// Mitsubishi GX Works2 project: PLC_2   PLC: Q04UDV

PROGRAM MAIN
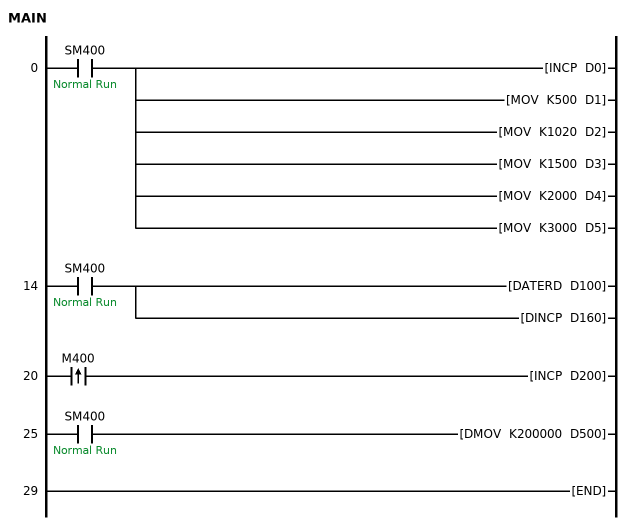
0     LD      SM400  ; Normal Run
      INCP    D0
      MOV     K500 D1
      MOV     K1020 D2
      MOV     K1500 D3
      MOV     K2000 D4
      MOV     K3000 D5
14    LD      SM400  ; Normal Run
      DATERD  D100
      DINCP   D160
20    LDP     M400
      INCP    D200
25    LD      SM400  ; Normal Run
      DMOV    K200000 D500
29    END
END_PROGRAM

PROGRAM LOSSCODE
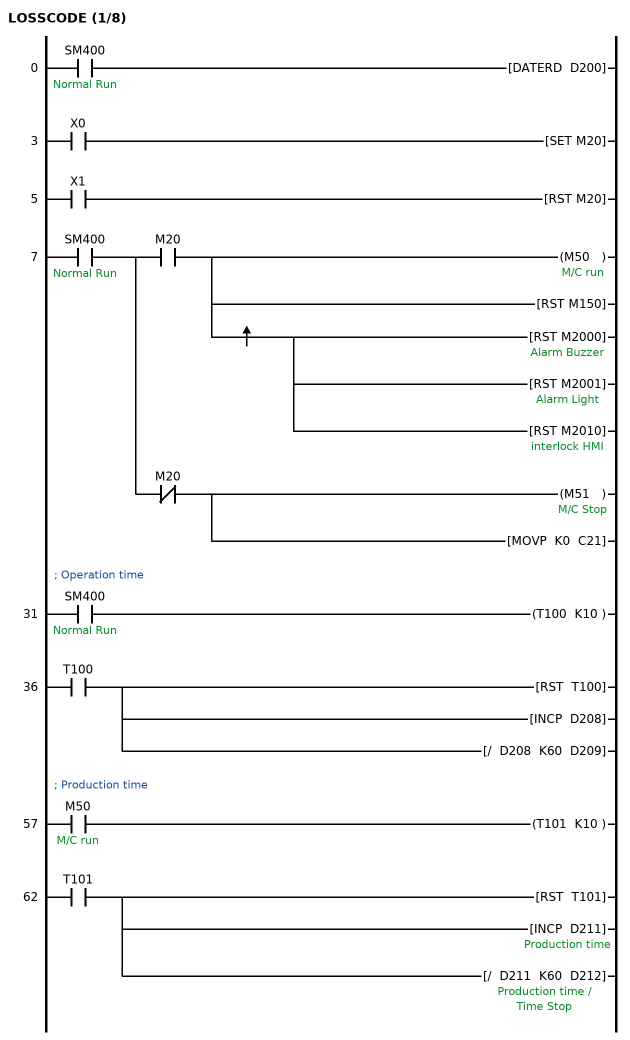
0     LD      SM400  ; Normal Run
      DATERD  D200
3     LD      X0
      SET     M20
5     LD      X1
      RST     M20
7     LD      SM400  ; Normal Run
      MPS
      AND     M20
      OUT     M50  ; M/C run
      RST     M150
      MEP
      RST     M2000  ; Alarm Buzzer
      RST     M2001  ; Alarm Light
      RST     M2010  ; interlock HMI
      MPP
      ANI     M20
      OUT     M51  ; M/C Stop
      MOVP    K0 C21
; Operation time
31    LD      SM400  ; Normal Run
      OUT     T100 K10
36    LD      T100
      RST     T100
      INCP    D208
      /       D208 K60 D209
; Production time
57    LD      M50  ; M/C run
      OUT     T101 K10
62    LD      T101
      RST     T101
      INCP    D211  ; Production time
      /       D211 K60 D212  ; Time Stop
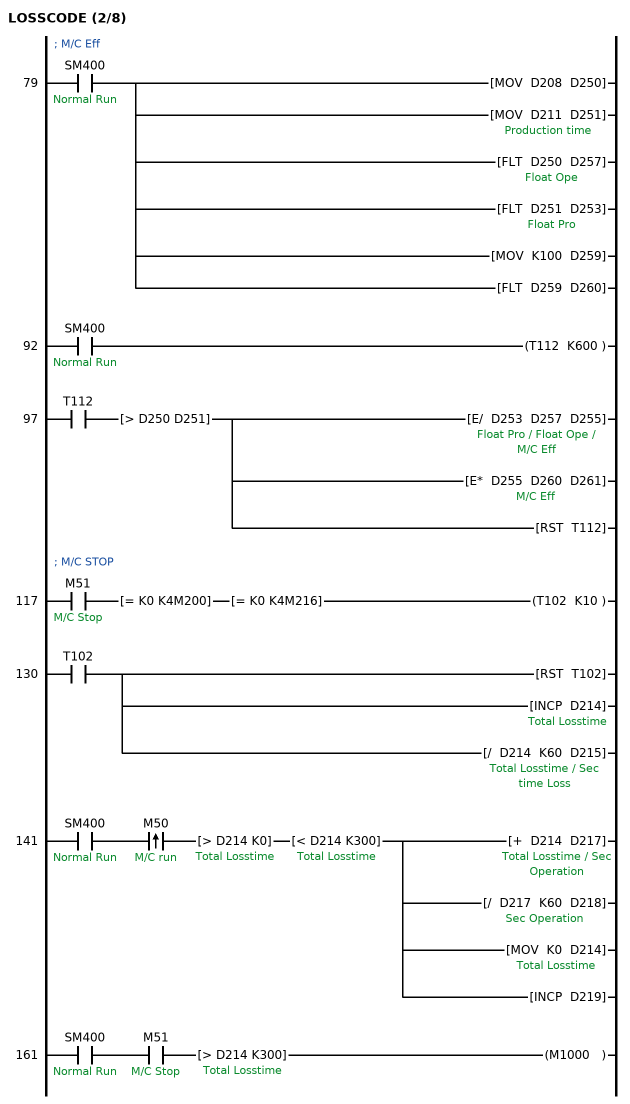
; M/C Eff
79    LD      SM400  ; Normal Run
      MOV     D208 D250
      MOV     D211 D251
      FLT     D250 D257  ; Float Ope
      FLT     D251 D253  ; Float Pro
      MOV     K100 D259
      FLT     D259 D260
92    LD      SM400  ; Normal Run
      OUT     T112 K600
97    LD      T112
      AND>    D250 D251
      E/      D253 D257 D255  ; M/C Eff
      E*      D255 D260 D261
      RST     T112
; M/C STOP
117   LD      M51  ; M/C Stop
      AND=    K0 K4M200
      AND=    K0 K4M216
      OUT     T102 K10
130   LD      T102
      RST     T102
      INCP    D214  ; Total Losstime
      /       D214 K60 D215  ; Sec time Loss
141   LD      SM400  ; Normal Run
      ANDP    M50  ; M/C run
      AND>    D214 K0  ; Total Losstime
      AND<    D214 K300  ; Total Losstime
      +       D214 D217  ; Sec Operation
      /       D217 K60 D218
      MOV     K0 D214
      INCP    D219
161   LD      SM400  ; Normal Run
      AND     M51  ; M/C Stop
      AND>    D214 K300  ; Total Losstime
      OUT     M1000
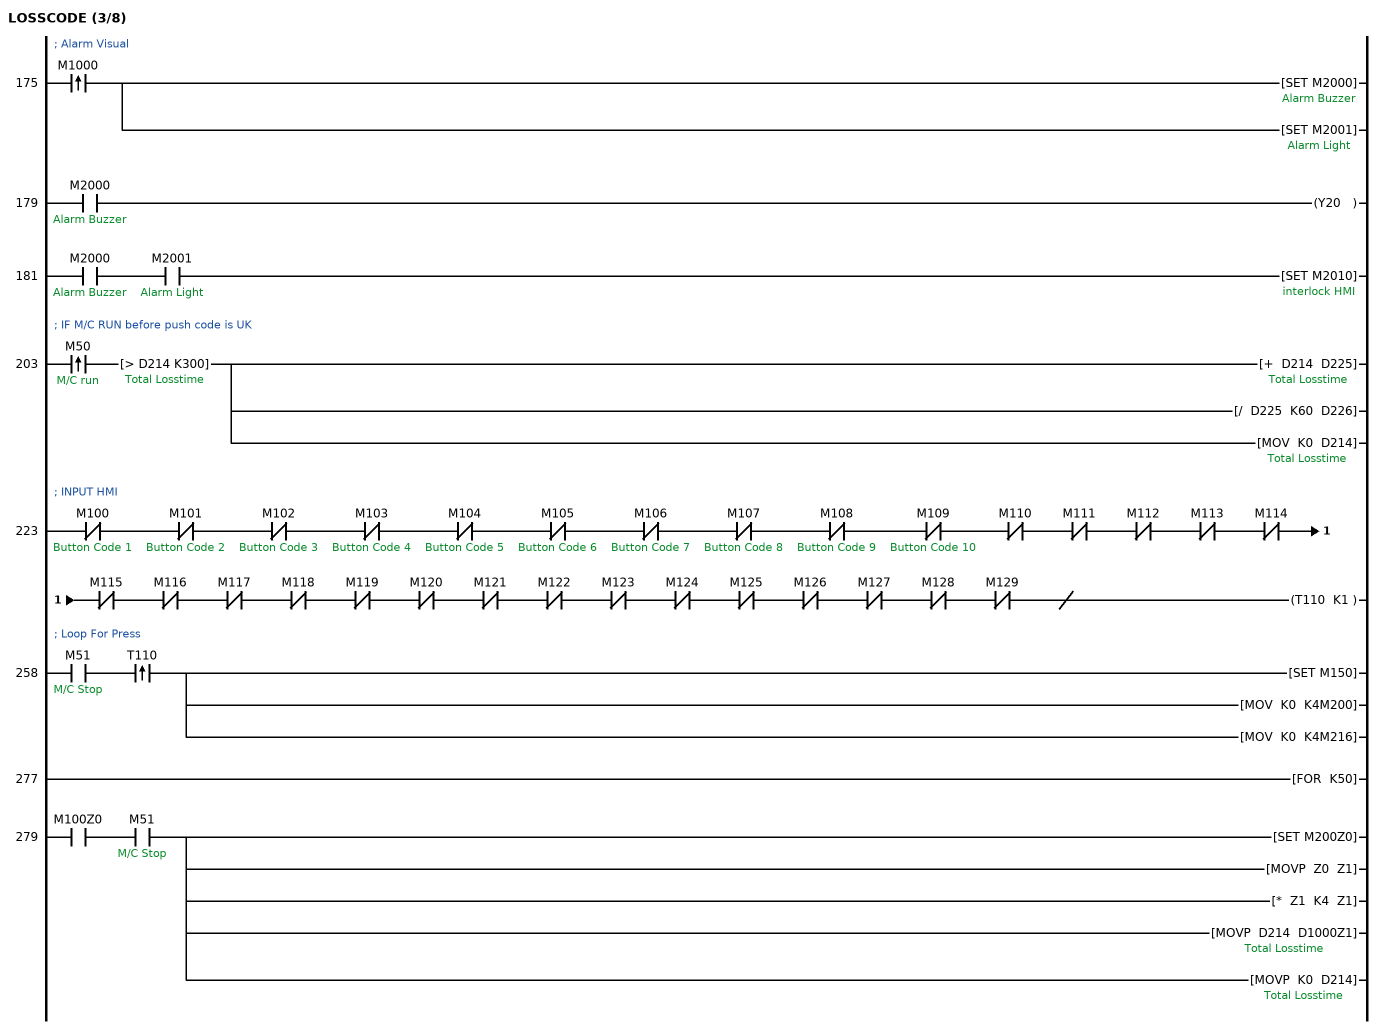
; Alarm Visual
175   LDP     M1000
      SET     M2000  ; Alarm Buzzer
      SET     M2001  ; Alarm Light
179   LD      M2000  ; Alarm Buzzer
      OUT     Y20
181   LD      M2000  ; Alarm Buzzer
      AND     M2001  ; Alarm Light
      SET     M2010  ; interlock HMI
; IF M/C RUN before push code is UK
203   LDP     M50  ; M/C run
      AND>    D214 K300  ; Total Losstime
      +       D214 D225
      /       D225 K60 D226
      MOV     K0 D214
; INPUT HMI
223   LDI     M100  ; Button Code 1
      ANI     M101  ; Button Code 2
      ANI     M102  ; Button Code 3
      ANI     M103  ; Button Code 4
      ANI     M104  ; Button Code 5
      ANI     M105  ; Button Code 6
      ANI     M106  ; Button Code 7
      ANI     M107  ; Button Code 8
      ANI     M108  ; Button Code 9
      ANI     M109  ; Button Code 10
      ANI     M110
      ANI     M111
      ANI     M112
      ANI     M113
      ANI     M114
      ANI     M115
      ANI     M116
      ANI     M117
      ANI     M118
      ANI     M119
      ANI     M120
      ANI     M121
      ANI     M122
      ANI     M123
      ANI     M124
      ANI     M125
      ANI     M126
      ANI     M127
      ANI     M128
      ANI     M129
      INV
      OUT     T110 K1
258   LD      M51  ; M/C Stop
      ANDP    T110
      SET     M150
      MOV     K0 K4M200
      MOV     K0 K4M216
; Loop For Press
277   FOR     K50
279   LD      M100Z0
      AND     M51  ; M/C Stop
      SET     M200Z0
      MOVP    Z0 Z1
      *       Z1 K4 Z1
      MOVP    D214 D1000Z1
      MOVP    K0 D214
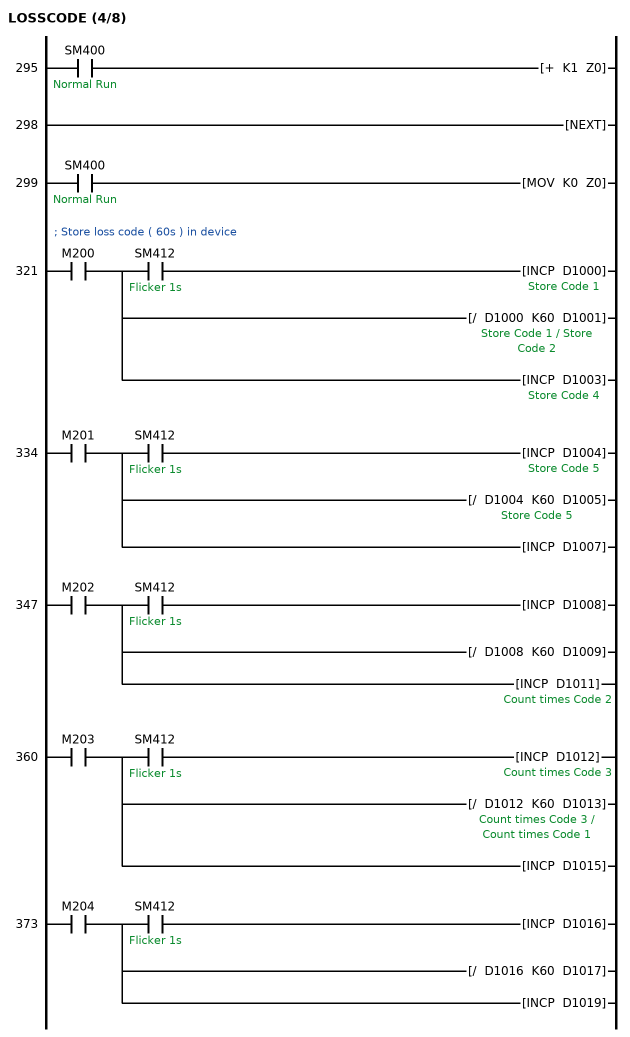
295   LD      SM400  ; Normal Run
      +       K1 Z0
298   NEXT
299   LD      SM400  ; Normal Run
      MOV     K0 Z0
; Store loss code ( 60s ) in device
321   LD      M200
      MPS
      AND     SM412  ; Flicker 1s
      INCP    D1000  ; Store Code 1
      MPP
      /       D1000 K60 D1001  ; Store Code 2
      INCP    D1003  ; Store Code 4
334   LD      M201
      MPS
      AND     SM412  ; Flicker 1s
      INCP    D1004  ; Store Code 5
      MPP
      /       D1004 K60 D1005
      INCP    D1007
347   LD      M202
      MPS
      AND     SM412  ; Flicker 1s
      INCP    D1008
      MPP
      /       D1008 K60 D1009
      INCP    D1011  ; Count times Code 2
360   LD      M203
      MPS
      AND     SM412  ; Flicker 1s
      INCP    D1012  ; Count times Code 3
      MPP
      /       D1012 K60 D1013  ; Count times Code 1
      INCP    D1015
373   LD      M204
      MPS
      AND     SM412  ; Flicker 1s
      INCP    D1016
      MPP
      /       D1016 K60 D1017
      INCP    D1019
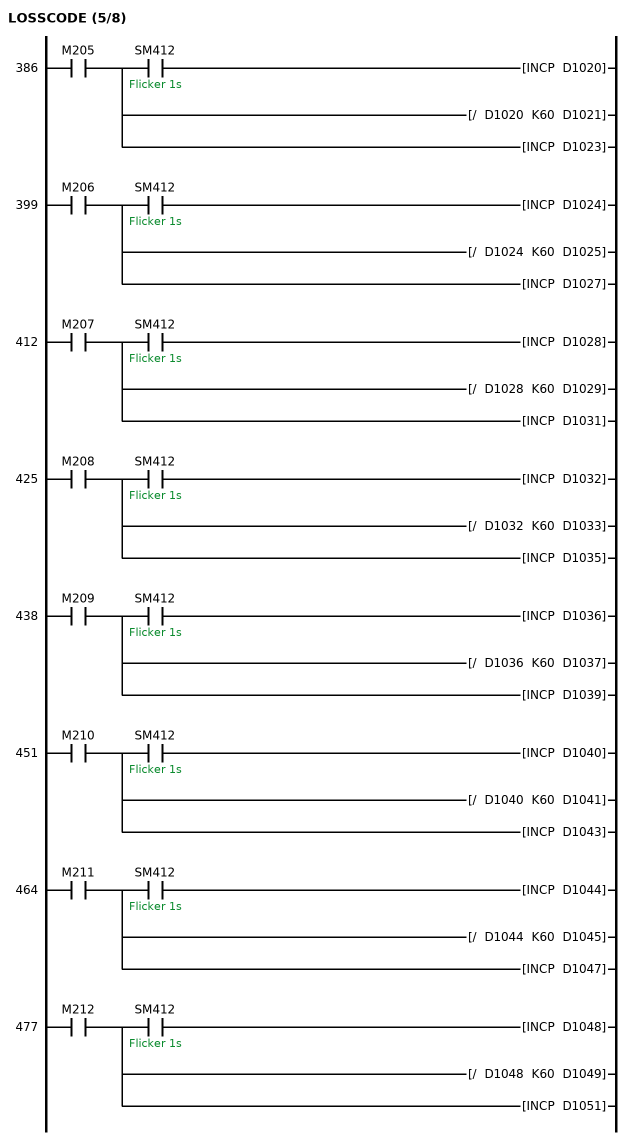
386   LD      M205
      MPS
      AND     SM412  ; Flicker 1s
      INCP    D1020
      MPP
      /       D1020 K60 D1021
      INCP    D1023
399   LD      M206
      MPS
      AND     SM412  ; Flicker 1s
      INCP    D1024
      MPP
      /       D1024 K60 D1025
      INCP    D1027
412   LD      M207
      MPS
      AND     SM412  ; Flicker 1s
      INCP    D1028
      MPP
      /       D1028 K60 D1029
      INCP    D1031
425   LD      M208
      MPS
      AND     SM412  ; Flicker 1s
      INCP    D1032
      MPP
      /       D1032 K60 D1033
      INCP    D1035
438   LD      M209
      MPS
      AND     SM412  ; Flicker 1s
      INCP    D1036
      MPP
      /       D1036 K60 D1037
      INCP    D1039
451   LD      M210
      MPS
      AND     SM412  ; Flicker 1s
      INCP    D1040
      MPP
      /       D1040 K60 D1041
      INCP    D1043
464   LD      M211
      MPS
      AND     SM412  ; Flicker 1s
      INCP    D1044
      MPP
      /       D1044 K60 D1045
      INCP    D1047
477   LD      M212
      MPS
      AND     SM412  ; Flicker 1s
      INCP    D1048
      MPP
      /       D1048 K60 D1049
      INCP    D1051
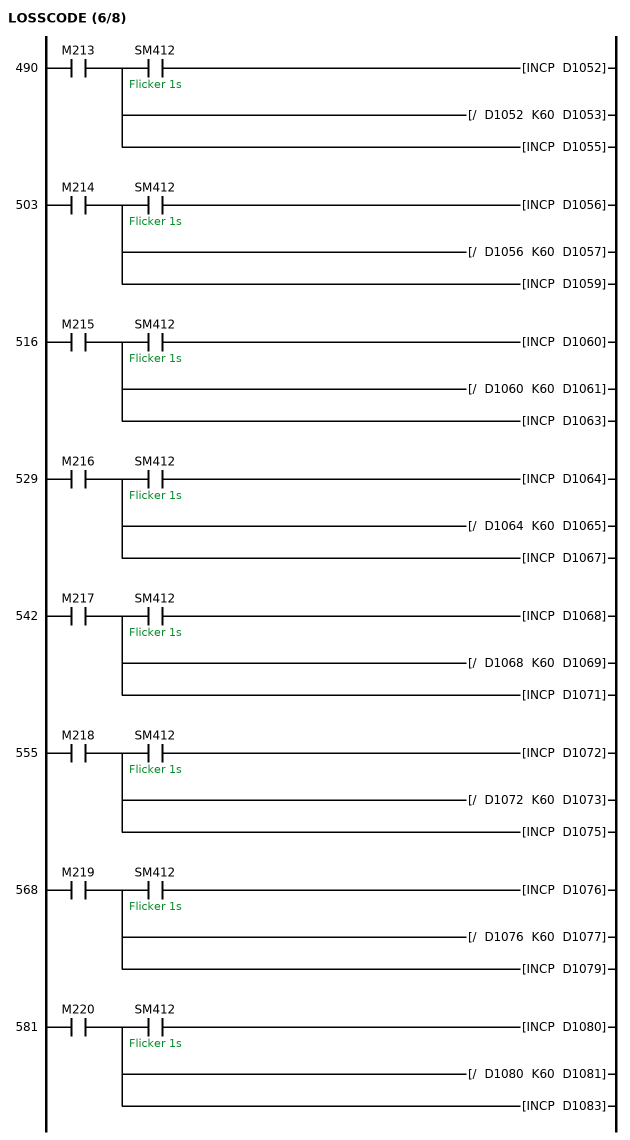
490   LD      M213
      MPS
      AND     SM412  ; Flicker 1s
      INCP    D1052
      MPP
      /       D1052 K60 D1053
      INCP    D1055
503   LD      M214
      MPS
      AND     SM412  ; Flicker 1s
      INCP    D1056
      MPP
      /       D1056 K60 D1057
      INCP    D1059
516   LD      M215
      MPS
      AND     SM412  ; Flicker 1s
      INCP    D1060
      MPP
      /       D1060 K60 D1061
      INCP    D1063
529   LD      M216
      MPS
      AND     SM412  ; Flicker 1s
      INCP    D1064
      MPP
      /       D1064 K60 D1065
      INCP    D1067
542   LD      M217
      MPS
      AND     SM412  ; Flicker 1s
      INCP    D1068
      MPP
      /       D1068 K60 D1069
      INCP    D1071
555   LD      M218
      MPS
      AND     SM412  ; Flicker 1s
      INCP    D1072
      MPP
      /       D1072 K60 D1073
      INCP    D1075
568   LD      M219
      MPS
      AND     SM412  ; Flicker 1s
      INCP    D1076
      MPP
      /       D1076 K60 D1077
      INCP    D1079
581   LD      M220
      MPS
      AND     SM412  ; Flicker 1s
      INCP    D1080
      MPP
      /       D1080 K60 D1081
      INCP    D1083
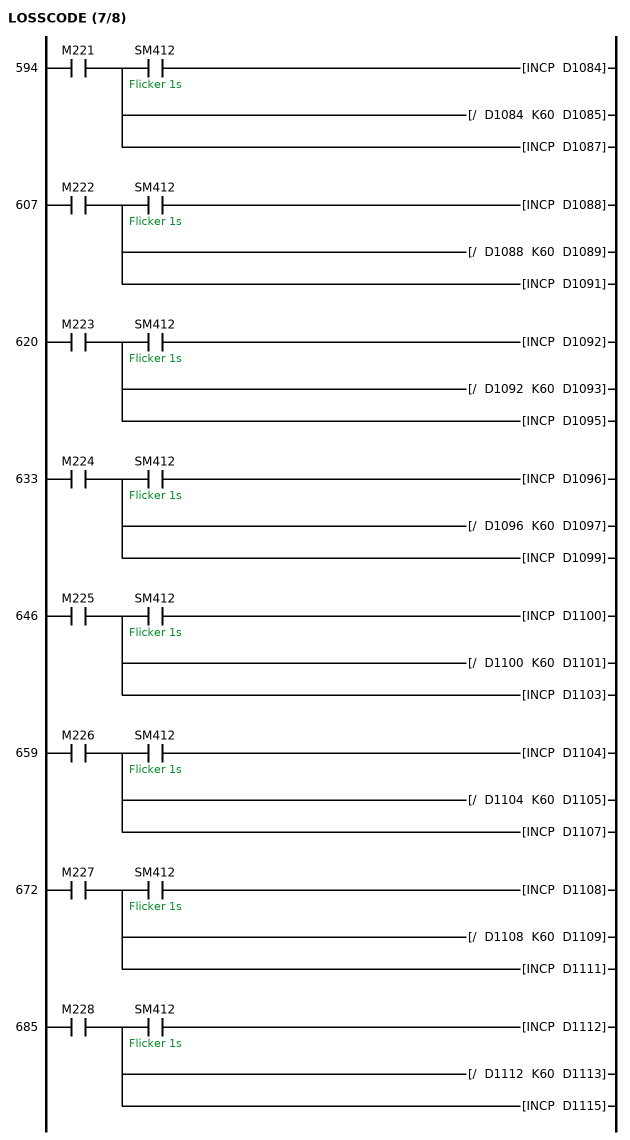
594   LD      M221
      MPS
      AND     SM412  ; Flicker 1s
      INCP    D1084
      MPP
      /       D1084 K60 D1085
      INCP    D1087
607   LD      M222
      MPS
      AND     SM412  ; Flicker 1s
      INCP    D1088
      MPP
      /       D1088 K60 D1089
      INCP    D1091
620   LD      M223
      MPS
      AND     SM412  ; Flicker 1s
      INCP    D1092
      MPP
      /       D1092 K60 D1093
      INCP    D1095
633   LD      M224
      MPS
      AND     SM412  ; Flicker 1s
      INCP    D1096
      MPP
      /       D1096 K60 D1097
      INCP    D1099
646   LD      M225
      MPS
      AND     SM412  ; Flicker 1s
      INCP    D1100
      MPP
      /       D1100 K60 D1101
      INCP    D1103
659   LD      M226
      MPS
      AND     SM412  ; Flicker 1s
      INCP    D1104
      MPP
      /       D1104 K60 D1105
      INCP    D1107
672   LD      M227
      MPS
      AND     SM412  ; Flicker 1s
      INCP    D1108
      MPP
      /       D1108 K60 D1109
      INCP    D1111
685   LD      M228
      MPS
      AND     SM412  ; Flicker 1s
      INCP    D1112
      MPP
      /       D1112 K60 D1113
      INCP    D1115
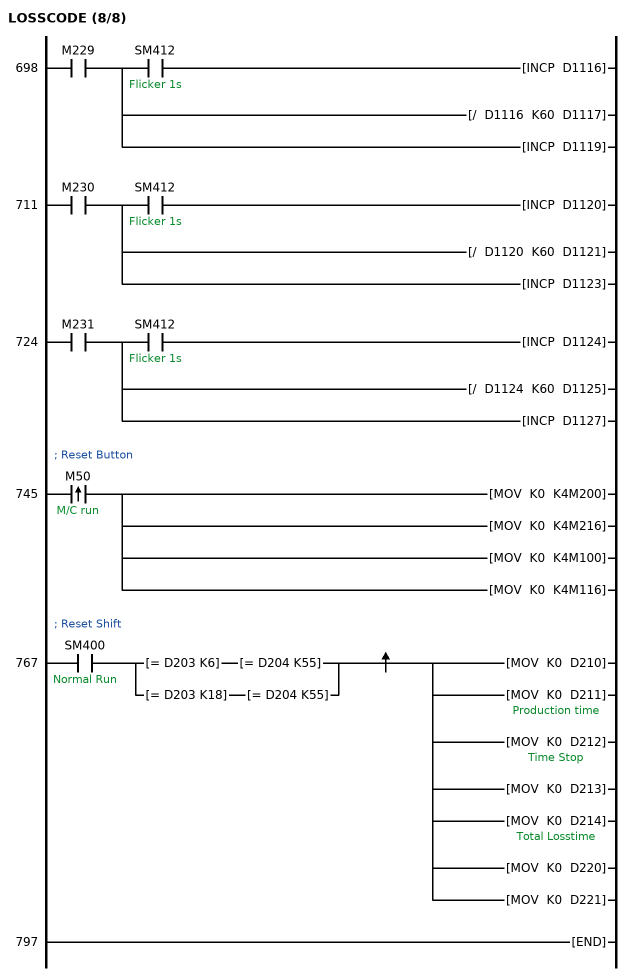
698   LD      M229
      MPS
      AND     SM412  ; Flicker 1s
      INCP    D1116
      MPP
      /       D1116 K60 D1117
      INCP    D1119
711   LD      M230
      MPS
      AND     SM412  ; Flicker 1s
      INCP    D1120
      MPP
      /       D1120 K60 D1121
      INCP    D1123
724   LD      M231
      MPS
      AND     SM412  ; Flicker 1s
      INCP    D1124
      MPP
      /       D1124 K60 D1125
      INCP    D1127
; Reset Button
745   LDP     M50  ; M/C run
      MOV     K0 K4M200
      MOV     K0 K4M216
      MOV     K0 K4M100
      MOV     K0 K4M116
; Reset Shift
767   LD      SM400  ; Normal Run
      LD=     D203 K6
      AND=    D204 K55
      LD=     D203 K18
      AND=    D204 K55
      ORB
      ANB
      MEP
      MOV     K0 D210
      MOV     K0 D211
      MOV     K0 D212
      MOV     K0 D213
      MOV     K0 D214
      MOV     K0 D220
      MOV     K0 D221
797   END
END_PROGRAM

// device comments not shown above
M47  ; Start
M1300  ; Button 1
M1301  ; Button 2
X28  ; Shutter 1
X29  ; Shutter 2
D216  ; Sec Production
D1002  ; Store Code 3
D1010  ; Count times Code 1
D1014  ; Count times Code 4
